{attribute 'GeneratedUsingTerminal: AMP8000-0030-0103-0103'}
{attribute addProperty BoxType "AMP8000-0030-0103-0103"}
{attribute addProperty Id "Ch_A_Target_positionAT %Q*DINT4Ch_A_Target_velocityAT %Q*DINT4"}
{attribute addProperty CRC "1177181981"}
{attribute addProperty Size "8"}
TYPE Ch_A_Interpolator_Outputs_462A5F1D EXTENDS OutputBase_10CEE7DE :
STRUCT
	{attribute addProperty Name "Ch_A_Target_position"}
	Ch_A_Target_position AT %Q* : DINT;
	{attribute addProperty Name "Ch_A_Target_velocity"}
	Ch_A_Target_velocity AT %Q* : DINT;
END_STRUCT
END_TYPE

(* stored: Version 1.2.0.0, ProductVersion 3.1.4024.11
   DUT Ch_A_Interpolator_Outputs_462A5F1D: Id {7d0e6f12-f05e-4f6d-af6f-23e03cf23a5f} *)
